FUNCTION_BLOCK FB_TOR_Rain EXTENDS FB_TOR_Base
//////////////////
//  Rain sensor system.
//////////////////

VAR_INPUT PERSISTENT
	// Parameters of the Object (instance/model specific) 
	ParamRainPerPulse				: REAL := 10 ; (* (mm) Number of mm of rain per pulse		*)
END_VAR

VAR_OUTPUT
	//Child objects
	
END_VAR

VAR_INPUT
	// I/O Inputs 		                                     				
    ParamVarHrWarning   			: REAL :=8 ;  // (mm) Max of raining before warning mm of rain for last hour --> Mean it is raining a lot  Defaut value 8       
    ParamVarDayWarning  			: REAL :=48;  // (mm )max of raining before warning mm of rain for last day  --> Mean it rained a lot during 1 day defaut value 48
	ParamVarMinAlarm				: REAL :=-5;  // (%)  Config : Minimal allowed Site Hygrometry 



	MesDataExd			: TOR_Rain;
END_VAR

VAR


	//M_ALARMMANAGEMENT VARIABLES//
		WarningDay					: BOOL;
		WarningHr					: BOOL;
		WarningValue				: BOOL;
	
	
	//M_Execute
		FB_AverageHr				: FB_Average; 	
	    FB_AverageDay               : FB_Average;
	    FB_AverageMonth             : FB_Average;
		CTUHr						: CTU;
		CTUDay						: CTU;
		CTUMonth					: CTU;
		Hour 						: INT;
		PluvioHr_Avg		        : REAL ; 
		PluvioDay_Avg		        : REAL ; 
		PluvioMonth_Avg		        : REAL ;     
		PluvioHr_Max		        : REAL;
		PluvioDay_Max		        : REAL ; 
		PluvioMonth_Max		        : REAL ; 
        PluvioHr					: REAL ; 
		PluvioDay					: REAL ; 
		PluvioMonth					: REAL ; 

	
	
END_VAR

METHOD M_AlarmManagement
//////////////////
// Manages Door sensor alarms and warnings
/////////////////

VAR 
	// Method local variables (reinitialized at each cycle) 
	FB_AlarmCodeManager : FB_AlarmCodeManager ; 
END_VAR
	WarningDay	:= PluvioDay >= ParamVarDayWarning;
	WarningHr	:= PluvioHr >= ParamVarHrWarning;
	WarningValue:= PluvioDay <= ParamVarMinAlarm OR PluvioHr <= ParamVarMinAlarm;

// ALARM CODE //
	FB_AlarmCodeManager(
 		bAlarm1			:= FALSE,    								// 
		bAlarm2			:= FALSE, 									// 
		bAlarm3			:= FALSE, 									// 
		bAlarm4			:= FALSE, 									// 
		bAlarm5			:= FALSE,     								//
		bAlarm6			:= FALSE,  									//
		bAlarm7			:= FALSE,  									//
		bAlarm8			:= FALSE,  									//
		bAlarm9			:= FALSE,    								// 
		bAlarm10		:= FALSE, 									// 
		bAlarm11		:= FALSE, 									// 
		bAlarm12		:= FALSE, 									// 
		bAlarm13		:= FALSE,									// 
		bAlarm14		:= FALSE,									// 
		bAlarm15		:= FALSE,									// 
		wAlarmCode		=>MesDataExd.MesData.MesAlarmCode);

// WARNING CODE //
	FB_AlarmCodeManager(
		bAlarm1			:= WarningHr,   							// Raining too hard 
		bAlarm2			:= WarningDay, 								// Raining a lot during one day
		bAlarm3			:= WarningValue, 							// Raining value not coherent
		bAlarm4			:= FALSE, 									// 
		bAlarm5			:= FALSE,    								// 
		bAlarm6			:= FALSE, 									// 
		bAlarm7			:= FALSE, 									// 
		bAlarm8			:= FALSE, 									// 
		bAlarm9			:= FALSE,    								// 
		bAlarm10		:= FALSE, 									// 
		bAlarm11		:= FALSE, 									// 
		bAlarm12		:= FALSE, 									// 
		bAlarm13		:= FALSE,									// 
		bAlarm14		:= FALSE,									// 
		bAlarm15		:= FALSE,									// 
		wAlarmCode		=>MesDataExd.MesData.MesWarningCode);

// EVENT CODE //
	FB_AlarmCodeManager(
		bAlarm1			:= MesDataExd.MesData.MesAlarmState, 		// 0.2mm of water falled
		bAlarm2			:= FALSE, 									// 
		bAlarm3			:= FALSE, 									// 
		bAlarm4			:= FALSE, 									// 
		bAlarm5			:= FALSE, 									// 
		bAlarm6			:= FALSE, 									// 
		bAlarm7			:= FALSE, 									// 
		bAlarm8			:= FALSE, 									// 
		bAlarm9			:= FALSE, 									// 
		bAlarm10		:= FALSE, 									// 
		bAlarm11		:= FALSE, 									// 
		bAlarm12		:= FALSE, 									// 
		bAlarm13		:= FALSE, 									// 
		bAlarm14		:= FALSE, 									//  
		bAlarm15		:= FALSE, 									//  
		wAlarmCode		=>MesDataExd.MesData.MesEventCode);
END_METHOD

METHOD M_Execute
//////////////////
//  Method Calls 
/////////////////

VAR 
	// Method local variables (reinitialized at each cycle) 
	
END_VAR
// EMULATOR I/O //

//MAIN CODE HERE
Hour 							:=CstCycleTime_G/1000/3600  ;                        

CTUHr   (CU:= MesDataExd.MesData.MesAlarmState , RESET :=  Hour MOD 1 = 0) ; 
CTUDay  (CU:= MesDataExd.MesData.MesAlarmState , RESET := Hour MOD 24 = 0 ) ; 
CTUMonth(CU:= MesDataExd.MesData.MesAlarmState , RESET := Hour MOD 24*30 = 0 ) ; 

PluvioHr_Max := SEL( Hour MOD 1 = 0  ,   PluvioHr_Max , PluvioHr_Max:= PluvioHr)  ; 
PluvioHr := CTUHr.CV * ParamRainPerPulse ; 

PluvioDay_Max := SEL( Hour MOD 24 = 0  ,   PluvioDay_Max , PluvioDay_Max:= PluvioDay)  ; 
PluvioDay := CTUDay.CV * ParamRainPerPulse ; 

PluvioMonth_Max := SEL( Hour MOD 24*30 = 0  ,   PluvioMonth_Max , PluvioMonth_Max:= PluvioMonth)  ; 
PluvioMonth := CTUMonth.CV * ParamRainPerPulse ; 


//FB_AverageHr(ValueIn:=PluvioHr_Max  , WindowDuration := 24*3600*1000 , ValueOut => PluvioHr_Avg) ; 
//FB_AverageDay(ValueIn:=PluvioDay_Max  , WindowDuration := 24*30*3600*1000 , ValueOut => PluvioDay_Avg) ; 
//FB_AverageMonth(ValueIn:=PluvioMonth_Max  , WindowDuration := 24*365*3600*1000 , ValueOut => PluvioMonth_Avg) ;
//EVALUATE

MesDataExd.MesRainFall_LastHour 	:= PluvioHr;
MesDataExd.MesRainFall_LastDay		:= PluvioDay;
MesDataExd.MesRainFall_LastMonth	:= PluvioMonth;
MesDataExd.AvgmmHour				:= PluvioHr_Avg;
MesDataExd.AvgmmDay					:= PluvioDay_Avg;
MesDataExd.AvgmmMonth				:= PluvioMonth_Avg;

SUPER^.M_Execute();
END_METHOD

METHOD M_StateManager
//////////////////
// Detect when fire occurs
/////////////////

VAR 
	// Method local variables (reinitialized at each cycle)
 	MesStateInterm1 : BOOL;
	MesStateInterm2 : BOOL;
END_VAR

IF ParamCableCutSecurity THEN
	MesStateInterm1 := NOT IN_MesState1_IO ; 
	MesStateInterm2 := NOT IN_MesState2_IO ; 
ELSE 
	MesStateInterm1 := IN_MesState1_IO;
	MesStateInterm2 := IN_MesState2_IO;
END_IF

IF ParamNbSensors = 1 THEN 
	MesStateInterm2 := MesStateInterm1 ;
END_IF

IF ParamAtleastOne THEN 
MesDataExd.MesData.MesAlarmState := MesStateInterm1 OR MesStateInterm2 ; 
ELSE
MesDataExd.MesData.MesAlarmState := MesStateInterm1 AND MesStateInterm2 ; 
END_IF

R_TRIGAlarm(CLK:= MesDataExd.MesData.MesAlarmState ) ; 
IF R_TRIGAlarm.Q THEN
	MesCountAlarm :=  MIN(MesCountAlarm + 1 ,4294967295 ) ; 
ELSIF IN_ResetCounter THEN 
	MesCountAlarm := 0 ; 
END_IF

MesDataExd.MesData.MesCountAlarm	:= MesCountAlarm ;
END_METHOD

END_FUNCTION_BLOCK

(* stored: Version 1.1.0.1, ProductVersion 3.1.4024.12
   POU FB_TOR_Rain: Id {cbf909a3-b333-4e53-b531-e0cd015bd491}, SpecialFunc None
   Method M_AlarmManagement: Id {ca46844c-04f7-4a0d-ac89-5dba98bd6ad2}
   Method M_Execute: Id {cf8b742a-c207-4559-abcd-732d2386b9d5}
   Method M_StateManager: Id {476a2809-d654-4084-ae69-e2a805cb5dee} *)
